FUNCTION_BLOCK FB_ConveyorExit_ST
VAR_INPUT
END_VAR
VAR_OUTPUT
END_VAR
VAR
	rTrigExit : Tc2_Standard.R_TRIG;
	ExitTrigger : BOOL;
	ExitEdgeDetected : BOOL;
	
	step : INT;
END_VAR
VAR_IN_OUT
	control_data : PlantAndCMs.Udt_PlantControl_Mode_1;
	
	control_data_vision : CM_Vision_UDT;
	control_data_Conveyor2 : CM_DO_UDT;
	
	control_data_sorter1 : CM_DO_UDT;
	control_data_sorter2 : CM_DO_UDT;
	control_data_sorter3 : CM_DO_UDT;
	
	control_data_atExit : CM_DIN_UDT;
END_VAR

rTrigExit(CLK := ExitTrigger, Q => ExitEdgeDetected);

CASE step OF 
	0 : // Init
	IF control_data.Auto_Out AND control_data.Startet_Out THEN
		step := 1;
	END_IF
	
	1: // wait for ready signal from ceonveyor entry
	
	
	IF GVL.readyForSorting THEN
		step := 2;
	END_IF
	
	2 : // check for GVL. which brick and act accordingly
	IF GVL.BLUE_TOP OR GVL.GREEN_TOP THEN
		step := 5;
	ELSIF GVL.BLUE_MIDDLE OR GVL.GREEN_MIDDLE THEN
		step := 10;
	ELSIF GVL.GREEN_BOTTOM OR GVL.BLUE_BOTTOM THEN
		step := 15;
		
	END_IF
	
	5:
		GVL.BLUE_TOP := FALSE;
		GVL.BLUE_BOTTOM := FALSE;
		GVL.BLUE_MIDDLE := FALSE;
		GVL.GREEN_TOP := FALSE;
		GVL.GREEN_BOTTOM := FALSE;
		GVL.GREEN_MIDDLE := FALSE;
		IF ExitEdgeDetected THEN
			step := 1;
			GVL.SortingDone := TRUE;
		END_IF
	10:
		GVL.BLUE_TOP := FALSE;
		GVL.BLUE_BOTTOM := FALSE;
		GVL.BLUE_MIDDLE := FALSE;
		GVL.GREEN_TOP := FALSE;
		GVL.GREEN_BOTTOM := FALSE;
		GVL.GREEN_MIDDLE := FALSE;
		IF ExitEdgeDetected THEN
			step := 1;
			GVL.SortingDone := TRUE;
		END_IF
	15:
		GVL.BLUE_TOP := FALSE;
		GVL.BLUE_BOTTOM := FALSE;
		GVL.BLUE_MIDDLE := FALSE;
		GVL.GREEN_TOP := FALSE;
		GVL.GREEN_BOTTOM := FALSE;
		GVL.GREEN_MIDDLE := FALSE;
		IF ExitEdgeDetected THEN
			step := 1;
			GVL.SortingDone := TRUE;
		END_IF
	 
END_CASE

ExitTrigger := control_data_atExit.AutoHigh; 

control_data_Sorter1.PO_HighCommand := step = 5;
control_data_sorter2.PO_HighCommand := step = 10;
control_data_sorter3.PO_HighCommand := step = 15;

control_data_Conveyor2.PO_HighCommand := step = 5 OR step = 10 OR step = 15;

END_FUNCTION_BLOCK

(* stored: Version 1.1.0.1, ProductVersion 3.1.4024.13
   POU FB_ConveyorExit_ST: Id {583597d2-ef3e-4a01-936b-7b8cd5bd8267}, SpecialFunc None *)
